TYPE BOXCAR :
STRUCT
	pX : REAL;
	pY : REAL;
	currentTrack : SINT;
	queueNum : DINT;
	carNum : SINT;
	
END_STRUCT
END_TYPE

(* stored: Version 1.1.0.1
   DUT BOXCAR: Id {903b4816-ae89-40d5-8573-3632da433666} *)
